SMOVL C00314 BC00314 V=166.7  +MOVJ EC00314
SMOVL C00315 BC00315 V=166.7  +MOVJ EC00315
SREFP 3 C00316 BC00316  +REFP EC00316
CALL JOB:SEARCH-R1-S13D
SET P024 P006
SFTON3D P024
SMOVL C00317 BC00317 V=166.7  +MOVJ EC00317
SMOVL C00318 BC00318 V=166.7  +MOVJ EC00318
SREFP 3 C00319 BC00319  +REFP EC00319
CALL JOB:SEARCH-R1-S13D
SET P024 P006
SFTON3D P024
SMOVL C00320 BC00320 V=166.7  +MOVJ EC00320
MOVL C00321 BC00321 V=1000.0  +MOVJ EC00321 VJ=100.00
MOVL C00322 BC00322 V=1000.0  +MOVJ EC00322 VJ=100.00
'EndPath S3665
'Path S4335
SFTOF3D
MOVJ C00323 BC00323 VJ=100.00  +MOVJ EC00323 VJ=100.00
MOVL C00324 BC00324 V=800.0  +MOVJ EC00324 VJ=100.00
SMOVL C00325 BC00325 V=166.7  +MOVJ EC00325
SREFP 3 C00326 BC00326  +REFP EC00326
CALL JOB:SEARCH-R1-S13D
SET P025 P006
SFTON3D P025
SMOVL C00327 BC00327 V=166.7  +MOVJ EC00327
SMOVL C00328 BC00328 V=166.7  +MOVJ EC00328
SREFP 3 C00329 BC00329  +REFP EC00329
CALL JOB:SEARCH-R1-S13D
SET P025 P006
SFTON3D P025
SMOVL C00330 BC00330 V=166.7  +MOVJ EC00330
SMOVL C00331 BC00331 V=166.7  +MOVJ EC00331
SREFP 3 C00332 BC00332  +REFP EC00332
CALL JOB:SEARCH-R1-S13D
SET P025 P006
SFTON3D P025
SMOVL C00333 BC00333 V=166.7  +MOVJ EC00333
MOVL C00334 BC00334 V=1000.0  +MOVJ EC00334 VJ=100.00
MOVL C00335 BC00335 V=1000.0  +MOVJ EC00335 VJ=100.00
'EndPath S4335
'Path S3666
SFTOF3D
MOVJ C00336 BC00336 VJ=100.00  +MOVJ EC00336 VJ=100.00
MOVL C00337 BC00337 V=800.0  +MOVJ EC00337 VJ=100.00
SMOVL C00338 BC00338 V=166.7  +MOVJ EC00338
SREFP 3 C00339 BC00339  +REFP EC00339
CALL JOB:SEARCH-R1-S13D
SET P026 P006
SFTON3D P026
SMOVL C00340 BC00340 V=166.7  +MOVJ EC00340
SREFP 3 C00341 BC00341  +REFP EC00341
CALL JOB:SEARCH-R1-S13D
SET P026 P006
SFTON3D P026
SMOVL C00342 BC00342 V=166.7  +MOVJ EC00342
MOVL C00343 BC00343 V=1000.0  +MOVJ EC00343 VJ=100.00
'EndPath S3666
MOVJ C00344 BC00344 VJ=100.00  +MOVJ EC00344 VJ=100.00
MOVJ C00345 BC00345 VJ=100.00  +MOVJ EC00345 VJ=100.00
'Path S3661
SFTOF3D
MOVJ C00346 BC00346 VJ=100.00  +MOVJ EC00346 VJ=100.00
MOVL C00347 BC00347 V=800.0  +MOVJ EC00347 VJ=100.00
SMOVL C00348 BC00348 V=166.7  +MOVJ EC00348
SREFP 3 C00349 BC00349  +REFP EC00349
CALL JOB:SEARCH-R1-S13D
SET P027 P006
SFTON3D P027
SMOVL C00350 BC00350 V=166.7  +MOVJ EC00350
SMOVL C00351 BC00351 V=166.7  +MOVJ EC00351
SREFP 3 C00352 BC00352  +REFP EC00352
CALL JOB:SEARCH-R1-S13D
SET P027 P006
SFTON3D P027
SMOVL C00353 BC00353 V=250.0  +MOVJ EC00353
SMOVL C00354 BC00354 V=166.7  +MOVJ EC00354
SREFP 3 C00355 BC00355  +REFP EC00355
CALL JOB:SEARCH-R1-S13D
SET P027 P006
SFTON3D P027
SMOVL C00356 BC00356 V=166.7  +MOVJ EC00356
MOVL C00357 BC00357 V=1000.0  +MOVJ EC00357 VJ=100.00
MOVL C00358 BC00358 V=1000.0  +MOVJ EC00358 VJ=100.00
'EndPath S3661
'Path S4336
SFTOF3D
MOVJ C00359 BC00359 VJ=100.00  +MOVJ EC00359 VJ=100.00
MOVL C00360 BC00360 V=800.0  +MOVJ EC00360 VJ=100.00
SMOVL C00361 BC00361 V=166.7  +MOVJ EC00361
SREFP 3 C00362 BC00362  +REFP EC00362
CALL JOB:SEARCH-R1-S13D
SET P028 P006
SFTON3D P028
SMOVL C00363 BC00363 V=166.7  +MOVJ EC00363
SREFP 3 C00364 BC00364  +REFP EC00364
CALL JOB:SEARCH-R1-S13D
SET P028 P006
SFTON3D P028
SMOVL C00365 BC00365 V=166.7  +MOVJ EC00365
MOVL C00366 BC00366 V=1000.0  +MOVJ EC00366 VJ=100.00
'EndPath S4336
MOVJ C00367 BC00367 VJ=100.00  +MOVJ EC00367 VJ=100.00
'Path S4879
SFTOF3D
MOVJ C00368 BC00368 VJ=100.00  +MOVJ EC00368 VJ=100.00
MOVL C00369 BC00369 V=800.0  +MOVJ EC00369 VJ=100.00
SMOVL C00370 BC00370 V=166.7  +MOVJ EC00370
SREFP 3 C00371 BC00371  +REFP EC00371
CALL JOB:SEARCH-R1-S13D
SET P060 P006
SFTON3D P060
SMOVL C00372 BC00372 V=166.7  +MOVJ EC00372
SMOVL C00373 BC00373 V=166.7  +MOVJ EC00373
SREFP 3 C00374 BC00374  +REFP EC00374
CALL JOB:SEARCH-R1-S13D
SET P060 P006
SFTON3D P060
SMOVL C00375 BC00375 V=166.7  +MOVJ EC00375
SMOVL C00376 BC00376 V=250.0  +MOVJ EC00376
SMOVL C00377 BC00377 V=166.7  +MOVJ EC00377
SREFP 3 C00378 BC00378  +REFP EC00378
CALL JOB:SEARCH-R1-S13D
SET P060 P006
SFTON3D P060
SMOVL C00379 BC00379 V=166.7  +MOVJ EC00379
MOVL C00380 BC00380 V=1000.0  +MOVJ EC00380 VJ=100.00
'EndPath S4879
MOVJ C00381 BC00381 VJ=100.00  +MOVJ EC00381 VJ=100.00
'Path S3664
SFTOF3D
COMM PAUSE
COMM MOVJ C00382 BC00382 VJ=100.00  +MOVJ EC00382 VJ=100.00
COMM MOVL C00383 BC00383 V=800.0  +MOVJ EC00383 VJ=100.00
COMM SMOVL C00384 BC00384 V=166.7  +MOVJ EC00384
COMM SREFP 3 C00385 BC00385  +REFP EC00385
COMM CALL JOB:SEARCH-R1-S13D
COMM SET P029 P006
COMM SFTON3D P029
COMM SMOVL C00386 BC00386 V=166.7  +MOVJ EC00386
COMM SREFP 3 C00387 BC00387  +REFP EC00387
COMM CALL JOB:SEARCH-R1-S13D
COMM SET P029 P006
COMM SFTON3D P029
COMM SMOVL C00388 BC00388 V=166.7  +MOVJ EC00388
COMM MOVL C00389 BC00389 V=1000.0  +MOVJ EC00389 VJ=100.00
COMM 'EndPath S3664
COMM 'Path S4337
COMM SFTOF3D
COMM MOVJ C00390 BC00390 VJ=100.00  +MOVJ EC00390 VJ=100.00
COMM MOVL C00391 BC00391 V=800.0  +MOVJ EC00391 VJ=100.00
COMM SMOVL C00392 BC00392 V=166.7  +MOVJ EC00392
COMM SREFP 3 C00393 BC00393  +REFP EC00393
COMM CALL JOB:SEARCH-R1-S13D
COMM SET P030 P006
COMM SFTON3D P030
COMM SMOVL C00394 BC00394 V=166.7  +MOVJ EC00394
COMM SREFP 3 C00395 BC00395  +REFP EC00395
COMM CALL JOB:SEARCH-R1-S13D
COMM SET P030 P006
COMM SFTON3D P030
COMM SMOVL C00396 BC00396 V=166.7  +MOVJ EC00396
COMM MOVL C00397 BC00397 V=800.0  +MOVJ EC00397 VJ=100.00
COMM MOVL C00398 BC00398 V=1000.0  +MOVJ EC00398 VJ=100.00
COMM 'EndPath S4337
MOVJ C00399 BC00399 VJ=100.00  +MOVJ EC00399 VJ=100.00
'Path S3663
SFTOF3D
MOVJ C00400 BC00400 VJ=100.00  +MOVJ EC00400 VJ=100.00
MOVL C00401 BC00401 V=800.0  +MOVJ EC00401 VJ=100.00
SMOVL C00402 BC00402 V=166.7  +MOVJ EC00402
SREFP 3 C00403 BC00403  +REFP EC00403
CALL JOB:SEARCH-R1-S13D
SET P031 P006
SFTON3D P031
SMOVL C00404 BC00404 V=166.7  +MOVJ EC00404
SREFP 3 C00405 BC00405  +REFP EC00405
CALL JOB:SEARCH-R1-S13D
SET P031 P006
SFTON3D P031
SMOVL C00406 BC00406 V=166.7  +MOVJ EC00406
SMOVL C00407 BC00407 V=166.7  +MOVJ EC00407
SREFP 3 C00408 BC00408  +REFP EC00408
CALL JOB:SEARCH-R1-S13D
SET P031 P006
SFTON3D P031
SMOVL C00409 BC00409 V=166.7  +MOVJ EC00409
MOVL C00410 BC00410 V=1000.0  +MOVJ EC00410 VJ=100.00
'EndPath S3663
MOVJ C00411 BC00411 VJ=100.00  +MOVJ EC00411 VJ=100.00
'Path S4338
SFTOF3D
MOVJ C00412 BC00412 VJ=100.00  +MOVJ EC00412 VJ=100.00
MOVL C00413 BC00413 V=800.0  +MOVJ EC00413 VJ=100.00
SMOVL C00414 BC00414 V=166.7  +MOVJ EC00414
SREFP 3 C00415 BC00415  +REFP EC00415
CALL JOB:SEARCH-R1-S13D
SET P032 P006
SFTON3D P032
SMOVL C00416 BC00416 V=166.7  +MOVJ EC00416
SREFP 3 C00417 BC00417  +REFP EC00417
CALL JOB:SEARCH-R1-S13D
SET P032 P006
SFTON3D P032
SMOVL C00418 BC00418 V=166.7  +MOVJ EC00418
SMOVL C00419 BC00419 V=166.7  +MOVJ EC00419
SREFP 3 C00420 BC00420  +REFP EC00420
CALL JOB:SEARCH-R1-S13D
SET P032 P006
SFTON3D P032
SMOVL C00421 BC00421 V=166.7  +MOVJ EC00421
MOVL C00422 BC00422 V=1000.0  +MOVJ EC00422 VJ=100.00
'EndPath S4338
MOVJ C00423 BC00423 VJ=100.00  +MOVJ EC00423 VJ=100.00
'Path S3662
SFTOF3D
MOVJ C00424 BC00424 VJ=100.00  +MOVJ EC00424 VJ=100.00
MOVL C00425 BC00425 V=800.0  +MOVJ EC00425 VJ=100.00
SMOVL C00426 BC00426 V=166.7  +MOVJ EC00426
SREFP 3 C00427 BC00427  +REFP EC00427
CALL JOB:SEARCH-R1-S13D
SET P033 P006
SFTON3D P033
SMOVL C00428 BC00428 V=166.7  +MOVJ EC00428
SREFP 3 C00429 BC00429  +REFP EC00429
CALL JOB:SEARCH-R1-S13D
SET P033 P006
SFTON3D P033
SMOVL C00430 BC00430 V=166.7  +MOVJ EC00430
MOVL C00431 BC00431 V=1000.0  +MOVJ EC00431 VJ=100.00
'EndPath S3662
'Path S4339
SFTOF3D
MOVJ C00432 BC00432 VJ=100.00  +MOVJ EC00432 VJ=100.00
MOVL C00433 BC00433 V=800.0  +MOVJ EC00433 VJ=100.00
SMOVL C00434 BC00434 V=166.7  +MOVJ EC00434
SREFP 3 C00435 BC00435  +REFP EC00435
CALL JOB:SEARCH-R1-S13D
SET P034 P006
SFTON3D P034
SMOVL C00436 BC00436 V=166.7  +MOVJ EC00436
SMOVL C00437 BC00437 V=166.7  +MOVJ EC00437
SREFP 3 C00438 BC00438  +REFP EC00438
CALL JOB:SEARCH-R1-S13D
SET P034 P006
SFTON3D P034
SMOVL C00439 BC00439 V=166.7  +MOVJ EC00439
SMOVL C00440 BC00440 V=166.7  +MOVJ EC00440
SREFP 3 C00441 BC00441  +REFP EC00441
CALL JOB:SEARCH-R1-S13D
SET P034 P006
SFTON3D P034
SMOVL C00442 BC00442 V=166.7  +MOVJ EC00442
MOVL C00443 BC00443 V=1000.0  +MOVJ EC00443 VJ=100.00
'EndPath S4339
MOVJ C00444 BC00444 VJ=100.00  +MOVJ EC00444 VJ=100.00
'Path W3667
SFTOF3D
SFTON3D P026
MOVJ C00445 BC00445 VJ=100.00  +MOVJ EC00445 VJ=100.00
SMOVL C00446 BC00446 V=800.0  +MOVJ EC00446
SREFP 1 C00447 BC00447  +REFP EC00447
SREFP 2 C00448 BC00448  +REFP EC00448
SMOVL C00449 BC00449 V=166.7 PL=0  +MOVJ EC00449
MACRO1 MJ#(0) ARGF21
ARCON
SWVON WEV#(100)
SMOVL C00450 BC00450 V=9.2  +MOVJ EC00450
SMOVL C00451 BC00451 V=9.2  +MOVJ EC00451
SMOVL C00452 BC00452 V=9.2  +MOVJ EC00452
ARCOF
SWVOF
SMOVL C00453 BC00453 V=800.0  +MOVJ EC00453
SMOVL C00454 BC00454 V=1000.0  +MOVJ EC00454
SFTOF3D
'EndPath W3667
MOVJ C00455 BC00455 VJ=100.00  +MOVJ EC00455 VJ=100.00
MOVJ C00456 BC00456 VJ=100.00  +MOVJ EC00456 VJ=100.00
'Path W3668
SSFTOF
SFTOF3D
SFTON3D P028
MOVJ C00457 BC00457 VJ=100.00  +MOVJ EC00457 VJ=100.00
SMOVL C00458 BC00458 V=800.0  +MOVJ EC00458
SREFP 1 C00459 BC00459  +REFP EC00459
SREFP 2 C00460 BC00460  +REFP EC00460
SMOVL C00461 BC00461 V=150.0 PL=0  +MOVJ EC00461
ARCON
SWVON WEV#(100)
SFTON3D P027
SMOVL C00462 BC00462 V=9.2  +MOVJ EC00462
SMOVL C00463 BC00463 V=9.2  +MOVJ EC00463
ARCOF
SWVOF
SMOVL C00464 BC00464 V=800.0  +MOVJ EC00464
SMOVL C00465 BC00465 V=1000.0  +MOVJ EC00465
SFTOF3D
'EndPath W3668
MOVJ C00466 BC00466 VJ=100.00  +MOVJ EC00466 VJ=100.00
COMM 'Path W4546
COMM PAUSE
COMM SFTOF3D
COMM SFTON3D P022
COMM MOVJ C00467 BC00467 VJ=100.00  +MOVJ EC00467 VJ=100.00
COMM SMOVL C00468 BC00468 V=800.0  +MOVJ EC00468
COMM SMOVL C00469 BC00469 V=150.0 PL=0  +MOVJ EC00469
COMM MACRO1 MJ#(0) ARGF9
COMM ARCON
COMM SWVON WEV#(10)
COMM SFTON3D P021
COMM SMOVL C00470 BC00470 V=10.0  +MOVJ EC00470
COMM ARCOF
COMM SWVOF
COMM SMOVL C00471 BC00471 V=800.0  +MOVJ EC00471
COMM SMOVL C00472 BC00472 V=1000.0  +MOVJ EC00472
COMM SFTOF3D
COMM 'EndPath W4546
COMM 'Path W4901
COMM SFTOF3D
SFTON3D P060
COMM MOVJ C00473 BC00473 VJ=100.00  +MOVJ EC00473 VJ=100.00
MOVJ C00474 BC00474 VJ=100.00  +MOVJ EC00474 VJ=100.00
MOVJ C00475 BC00475 VJ=100.00  +MOVJ EC00475 VJ=100.00
SMOVL C00476 BC00476 V=800.0  +MOVJ EC00476
SMOVL C00477 BC00477 V=150.0 PL=0  +MOVJ EC00477
MACRO1 MJ#(0) ARGF14
ARCON
SMOVL C00478 BC00478 V=10.8  +MOVJ EC00478
ARCOF
SMOVL C00479 BC00479 V=800.0  +MOVJ EC00479
SFTOF3D
'EndPath W4901
'Path W4880
SFTOF3D
SFTON3D P060
SMOVL C00480 BC00480 V=800.0  +MOVJ EC00480
SMOVL C00481 BC00481 V=150.0 PL=0  +MOVJ EC00481
ARCON
SMOVL C00482 BC00482 V=10.0  +MOVJ EC00482
SMOVL C00483 BC00483 V=10.0  +MOVJ EC00483
SMOVL C00484 BC00484 V=10.0  +MOVJ EC00484
ARCOF
SMOVL C00485 BC00485 V=800.0  +MOVJ EC00485
SMOVL C00486 BC00486 V=1000.0  +MOVJ EC00486
SFTOF3D
'EndPath W4880
MOVJ C00487 BC00487 VJ=100.00  +MOVJ EC00487 VJ=100.00
COMM PAUSE
COMM MOVJ C00488 BC00488 VJ=100.00  +MOVJ EC00488 VJ=100.00
COMM 'Path W4548
COMM SFTOF3D
COMM SFTON3D P030
COMM MOVJ C00489 BC00489 VJ=100.00  +MOVJ EC00489 VJ=100.00
COMM SMOVL C00490 BC00490 V=800.0  +MOVJ EC00490
COMM SMOVL C00491 BC00491 V=150.0 PL=0  +MOVJ EC00491
COMM MACRO1 MJ#(0) ARGF9
COMM ARCON
COMM SFTON3D P029
COMM SMOVL C00492 BC00492 V=10.0  +MOVJ EC00492
COMM SMOVL C00493 BC00493 V=10.0  +MOVJ EC00493
COMM ARCOF
COMM SMOVL C00494 BC00494 V=800.0  +MOVJ EC00494
COMM SMOVL C00495 BC00495 V=1000.0  +MOVJ EC00495
COMM SFTOF3D
COMM 'EndPath W4548
COMM MOVJ C00496 BC00496 VJ=100.00  +MOVJ EC00496 VJ=100.00
MOVJ C00497 BC00497 VJ=100.00  +MOVJ EC00497 VJ=100.00
'Path W3671
SFTOF3D
SFTON3D P033
MOVJ C00498 BC00498 VJ=100.00  +MOVJ EC00498 VJ=100.00
SMOVL C00499 BC00499 V=800.0  +MOVJ EC00499
SMOVL C00500 BC00500 V=166.7 PL=0  +MOVJ EC00500
MACRO1 MJ#(0) ARGF14
ARCON
SMOVL C00501 BC00501 V=9.2  +MOVJ EC00501
SFTON3D P034
SMOVL C00502 BC00502 V=9.2  +MOVJ EC00502
SMOVL C00503 BC00503 V=9.2  +MOVJ EC00503
ARCOF
SMOVL C00504 BC00504 V=800.0  +MOVJ EC00504
SMOVL C00505 BC00505 V=1000.0  +MOVJ EC00505
SFTOF3D
'EndPath W3671
MOVJ C00506 BC00506 VJ=100.00  +MOVJ EC00506 VJ=100.00
'Path W3672
SFTOF3D
SFTON3D P024
MOVJ C00507 BC00507 VJ=100.00  +MOVJ EC00507 VJ=100.00
SMOVL C00508 BC00508 V=800.0  +MOVJ EC00508
SMOVL C00509 BC00509 V=166.7 PL=0  +MOVJ EC00509
ARCON
SMOVL C00510 BC00510 V=9.2  +MOVJ EC00510
SFTON3D P025
SMOVL C00511 BC00511 V=9.2  +MOVJ EC00511
SMOVL C00512 BC00512 V=9.2  +MOVJ EC00512
ARCOF
SMOVL C00513 BC00513 V=800.0  +MOVJ EC00513
SMOVL C00514 BC00514 V=1000.0  +MOVJ EC00514
SFTOF3D
'EndPath W3672
MOVJ C00515 BC00515 VJ=100.00  +MOVJ EC00515 VJ=100.00
'Path W3673
SFTOF3D
SFTON3D P032
MOVJ C00516 BC00516 VJ=100.00  +MOVJ EC00516 VJ=100.00
SMOVL C00517 BC00517 V=800.0  +MOVJ EC00517
SMOVL C00518 BC00518 V=166.7 PL=0  +MOVJ EC00518
ARCON
SMOVL C00519 BC00519 V=9.2  +MOVJ EC00519
SFTON3D P031
SMOVL C00520 BC00520 V=9.2  +MOVJ EC00520
SMOVL C00521 BC00521 V=9.2  +MOVJ EC00521
ARCOF
SMOVL C00522 BC00522 V=800.0  +MOVJ EC00522
SMOVL C00523 BC00523 V=1000.0  +MOVJ EC00523
SFTOF3D
'EndPath W3673
MOVJ C00524 BC00524 VJ=100.00  +MOVJ EC00524 VJ=100.00
'
MOVJ C00525 BC00525 VJ=100.00  +MOVJ EC00525 VJ=100.00
JUMP *VV
MOVJ C00526 BC00526 VJ=100.00  +MOVJ EC00526 VJ=100.00
'Path W3680
SFTOF3D
SFTON3D P023
MOVJ C00527 BC00527 VJ=100.00  +MOVJ EC00527 VJ=100.00
SMOVL C00528 BC00528 V=800.0  +MOVJ EC00528
SMOVL C00529 BC00529 V=166.7 PL=0  +MOVJ EC00529
SMOVL C00530 BC00530 V=10.0  +MOVJ EC00530
SMOVL C00531 BC00531 V=33.3  +MOVJ EC00531
SMOVL C00532 BC00532 V=33.3  +MOVJ EC00532
SMOVL C00533 BC00533 V=33.3  +MOVJ EC00533
SMOVL C00534 BC00534 V=10.0  +MOVJ EC00534
SMOVL C00535 BC00535 V=10.0  +MOVJ EC00535
SMOVL C00536 BC00536 V=10.0  +MOVJ EC00536
SMOVL C00537 BC00537 V=10.0  +MOVJ EC00537
SMOVL C00538 BC00538 V=10.0  +MOVJ EC00538
ARCOF
SMOVL C00539 BC00539 V=800.0  +MOVJ EC00539
SMOVL C00540 BC00540 V=1000.0  +MOVJ EC00540
SFTOF3D
'EndPath W3680
'Path W3681
*VV
SFTOF3D
SFTON3D P023
MOVJ C00541 BC00541 VJ=100.00  +MOVJ EC00541 VJ=100.00
SMOVL C00542 BC00542 V=800.0  +MOVJ EC00542
MACRO1 MJ#(0) ARGF9
SMOVL C00543 BC00543 V=166.7 PL=0  +MOVJ EC00543
COMM SMOVL C00544 BC00544 V=150.0 PL=0  +MOVJ EC00544
COMM MACRO1 MJ#(0) ARGF9
COMM ARCON
COMM SMOVL C00545 BC00545 V=8.3  +MOVJ EC00545
COMM SMOVL C00546 BC00546 V=8.3  +MOVJ EC00546
COMM SMOVL C00547 BC00547 V=8.3  +MOVJ EC00547
ARCON
SMOVL C00548 BC00548 V=8.3  +MOVJ EC00548
SMOVL C00549 BC00549 V=8.3  +MOVJ EC00549
SMOVL C00550 BC00550 V=8.3  +MOVJ EC00550
SMOVL C00551 BC00551 V=8.3  +MOVJ EC00551
SMOVL C00552 BC00552 V=8.3  +MOVJ EC00552
SMOVL C00553 BC00553 V=8.3  +MOVJ EC00553
ARCOF
SMOVL C00554 BC00554 V=800.0  +MOVJ EC00554
SMOVL C00555 BC00555 V=1000.0  +MOVJ EC00555
SFTOF3D
'EndPath W3681
'Down
MOVJ C00556 BC00556 VJ=100.00  +MOVJ EC00556 VJ=100.00
CALL JOB:CLEAN-R1_KM_3P
'1
MOVJ C00557 BC00557 VJ=100.00  +MOVJ EC00557 VJ=100.00
MOVJ C00558 BC00558 VJ=100.00  +MOVJ EC00558 VJ=100.00
MOVJ C00559 BC00559 VJ=100.00  +MOVJ EC00559 VJ=100.00
'Path S4334
SFTOF3D
MOVJ C00560 BC00560 VJ=100.00  +MOVJ EC00560 VJ=100.00
MOVL C00561 BC00561 V=800.0  +MOVJ EC00561 VJ=100.00
SMOVL C00562 BC00562 V=166.7  +MOVJ EC00562
SREFP 3 C00563 BC00563  +REFP EC00563
CALL JOB:SEARCH-R1-S13D
SET P048 P006
SFTON3D P048
SMOVL C00564 BC00564 V=166.7  +MOVJ EC00564
SMOVL C00565 BC00565 V=166.7  +MOVJ EC00565
SREFP 3 C00566 BC00566  +REFP EC00566
CALL JOB:SEARCH-R1-S13D
SET P048 P006
SFTON3D P048
SMOVL C00567 BC00567 V=166.7  +MOVJ EC00567
MOVL C00568 BC00568 V=1000.0  +MOVJ EC00568 VJ=100.00
'EndPath S4334
'Path S4335
SFTOF3D
MOVJ C00569 BC00569 VJ=100.00  +MOVJ EC00569 VJ=100.00
MOVL C00570 BC00570 V=800.0  +MOVJ EC00570 VJ=100.00
SMOVL C00571 BC00571 V=166.7  +MOVJ EC00571
SREFP 3 C00572 BC00572  +REFP EC00572
CALL JOB:SEARCH-R1-S13D
SET P047 P006
SFTON3D P047
SMOVL C00573 BC00573 V=250.0  +MOVJ EC00573
SMOVL C00574 BC00574 V=166.7  +MOVJ EC00574
SREFP 3 C00575 BC00575  +REFP EC00575
CALL JOB:SEARCH-R1-S13D
SET P047 P006
SFTON3D P047
SMOVL C00576 BC00576 V=166.7  +MOVJ EC00576
MOVL C00577 BC00577 V=1000.0  +MOVJ EC00577 VJ=100.00
'EndPath S4335
MOVJ C00578 BC00578 VJ=100.00  +MOVJ EC00578 VJ=100.00
MOVJ C00579 BC00579 VJ=100.00  +MOVJ EC00579 VJ=100.00
MOVJ C00580 BC00580 VJ=100.00  +MOVJ EC00580 VJ=100.00
MOVJ C00581 BC00581 VJ=100.00  +MOVJ EC00581 VJ=100.00
'Path S4336
SFTOF3D
MOVJ C00582 BC00582 VJ=100.00  +MOVJ EC00582 VJ=100.00
MOVL C00583 BC00583 V=800.0  +MOVJ EC00583 VJ=100.00
SMOVL C00584 BC00584 V=166.7  +MOVJ EC00584
SREFP 3 C00585 BC00585  +REFP EC00585
CALL JOB:SEARCH-R1-S13D
SET P046 P006
SFTON3D P046
SMOVL C00586 BC00586 V=250.0  +MOVJ EC00586
SMOVL C00587 BC00587 V=166.7  +MOVJ EC00587
SREFP 3 C00588 BC00588  +REFP EC00588
CALL JOB:SEARCH-R1-S13D
SET P046 P006
SFTON3D P046
SMOVL C00589 BC00589 V=166.7  +MOVJ EC00589
MOVL C00590 BC00590 V=1000.0  +MOVJ EC00590 VJ=100.00
'EndPath S4336
'Path S4337
SFTOF3D
MOVJ C00591 BC00591 VJ=100.00  +MOVJ EC00591 VJ=100.00
MOVL C00592 BC00592 V=800.0  +MOVJ EC00592 VJ=100.00
SMOVL C00593 BC00593 V=166.7  +MOVJ EC00593
SREFP 3 C00594 BC00594  +REFP EC00594
CALL JOB:SEARCH-R1-S13D
SET P050 P006
SFTON3D P050
SMOVL C00595 BC00595 V=166.7  +MOVJ EC00595
SREFP 3 C00596 BC00596  +REFP EC00596
CALL JOB:SEARCH-R1-S13D
SET P050 P006
SFTON3D P050
SMOVL C00597 BC00597 V=166.7  +MOVJ EC00597
MOVL C00598 BC00598 V=1000.0  +MOVJ EC00598 VJ=100.00
'EndPath S4337
'Path S4338
SFTOF3D
MOVJ C00599 BC00599 VJ=100.00  +MOVJ EC00599 VJ=100.00
MOVL C00600 BC00600 V=666.7  +MOVJ EC00600 VJ=100.00
SMOVL C00601 BC00601 V=166.7  +MOVJ EC00601
SREFP 3 C00602 BC00602  +REFP EC00602
CALL JOB:SEARCH-R1-S13D
SET P051 P006
SFTON3D P051
SMOVL C00603 BC00603 V=166.7  +MOVJ EC00603
SREFP 3 C00604 BC00604  +REFP EC00604
CALL JOB:SEARCH-R1-S13D
SET P051 P006
SFTON3D P051
SMOVL C00605 BC00605 V=166.7  +MOVJ EC00605
SMOVL C00606 BC00606 V=166.7  +MOVJ EC00606
SMOVL C00607 BC00607 V=133.3  +MOVJ EC00607
SREFP 3 C00608 BC00608  +REFP EC00608
CALL JOB:SEARCH-R1-S13D
SET P051 P006
SFTON3D P051
SMOVL C00609 BC00609 V=250.0  +MOVJ EC00609
SMOVL C00610 BC00610 V=500.0  +MOVJ EC00610
'EndPath S4338
'Path S4339
SFTOF3D
MOVJ C00611 BC00611 VJ=100.00  +MOVJ EC00611 VJ=100.00
MOVL C00612 BC00612 V=800.0  +MOVJ EC00612 VJ=100.00
SMOVL C00613 BC00613 V=166.7  +MOVJ EC00613
SREFP 3 C00614 BC00614  +REFP EC00614
CALL JOB:SEARCH-R1-S13D
SET P045 P006
SFTON3D P045
SMOVL C00615 BC00615 V=250.0  +MOVJ EC00615
SMOVL C00616 BC00616 V=166.7  +MOVJ EC00616
SREFP 3 C00617 BC00617  +REFP EC00617
CALL JOB:SEARCH-R1-S13D
SET P045 P006
SFTON3D P045
SMOVL C00618 BC00618 V=166.7  +MOVJ EC00618
MOVL C00619 BC00619 V=1000.0  +MOVJ EC00619 VJ=100.00
'EndPath S4339
'Path S4340
SFTOF3D
MOVJ C00620 BC00620 VJ=100.00  +MOVJ EC00620 VJ=100.00
MOVL C00621 BC00621 V=800.0  +MOVJ EC00621 VJ=100.00
SMOVL C00622 BC00622 V=166.7  +MOVJ EC00622
SREFP 3 C00623 BC00623  +REFP EC00623
CALL JOB:SEARCH-R1-S13D
SET P044 P006
SFTON3D P044
SMOVL C00624 BC00624 V=250.0  +MOVJ EC00624
SMOVL C00625 BC00625 V=166.7  +MOVJ EC00625
SREFP 3 C00626 BC00626  +REFP EC00626
CALL JOB:SEARCH-R1-S13D
SET P044 P006
SFTON3D P044
SMOVL C00627 BC00627 V=166.7  +MOVJ EC00627
MOVL C00628 BC00628 V=1000.0  +MOVJ EC00628 VJ=100.00
'EndPath S4340
'Path S4341
SFTOF3D
MOVJ C00629 BC00629 VJ=100.00  +MOVJ EC00629 VJ=100.00
MOVL C00630 BC00630 V=800.0  +MOVJ EC00630 VJ=100.00
SMOVL C00631 BC00631 V=166.7  +MOVJ EC00631
SREFP 3 C00632 BC00632  +REFP EC00632
CALL JOB:SEARCH-R1-S13D
SET P049 P006
SFTON3D P049
SMOVL C00633 BC00633 V=166.7  +MOVJ EC00633
SMOVL C00634 BC00634 V=166.7  +MOVJ EC00634
SREFP 3 C00635 BC00635  +REFP EC00635
CALL JOB:SEARCH-R1-S13D
SET P049 P006
SFTON3D P049
SMOVL C00636 BC00636 V=166.7  +MOVJ EC00636
MOVL C00637 BC00637 V=1000.0  +MOVJ EC00637 VJ=100.00
'EndPath S4341
MOVJ C00638 BC00638 VJ=100.00  +MOVJ EC00638 VJ=100.00
MOVJ C00639 BC00639 VJ=100.00  +MOVJ EC00639 VJ=100.00
'Path S4342
SFTOF3D
MOVJ C00640 BC00640 VJ=100.00  +MOVJ EC00640 VJ=100.00
MOVL C00641 BC00641 V=800.0  +MOVJ EC00641 VJ=100.00
SMOVL C00642 BC00642 V=166.7  +MOVJ EC00642
SREFP 3 C00643 BC00643  +REFP EC00643
CALL JOB:SEARCH-R1-S13D
SET P043 P006
SFTON3D P043
SMOVL C00644 BC00644 V=166.7  +MOVJ EC00644
SMOVL C00645 BC00645 V=166.7  +MOVJ EC00645
SREFP 3 C00646 BC00646  +REFP EC00646
CALL JOB:SEARCH-R1-S13D
SET P043 P006
SFTON3D P043
SMOVL C00647 BC00647 V=166.7  +MOVJ EC00647
MOVL C00648 BC00648 V=1000.0  +MOVJ EC00648 VJ=100.00
'EndPath S4342
'Path S4343
SFTOF3D
MOVJ C00649 BC00649 VJ=100.00  +MOVJ EC00649 VJ=100.00
MOVL C00650 BC00650 V=800.0  +MOVJ EC00650 VJ=100.00
SMOVL C00651 BC00651 V=166.7  +MOVJ EC00651
SREFP 3 C00652 BC00652  +REFP EC00652
CALL JOB:SEARCH-R1-S13D
SET P042 P006
SFTON3D P042
SMOVL C00653 BC00653 V=250.0  +MOVJ EC00653
SMOVL C00654 BC00654 V=166.7  +MOVJ EC00654
SREFP 3 C00655 BC00655  +REFP EC00655
CALL JOB:SEARCH-R1-S13D
SET P042 P006
SFTON3D P042
SMOVL C00656 BC00656 V=166.7  +MOVJ EC00656
MOVL C00657 BC00657 V=1000.0  +MOVJ EC00657 VJ=100.00
'EndPath S4343
MOVJ C00658 BC00658 VJ=100.00  +MOVJ EC00658 VJ=100.00
'
'Path W4344
SFTOF3D
SFTON3D P051
MOVJ C00659 BC00659 VJ=60.00  +MOVJ EC00659 VJ=20.00
SMOVL C00660 BC00660 V=500.0  +MOVJ EC00660
SMOVL C00661 BC00661 V=166.7 PL=0  +MOVJ EC00661
MACRO1 MJ#(0) ARGF14
ARCON
SMOVL C00662 BC00662 V=8.3  +MOVJ EC00662
ARCOF
SMOVL C00663 BC00663 V=800.0  +MOVJ EC00663
SMOVL C00664 BC00664 V=150.0  +MOVJ EC00664
ARCON
SMOVL C00665 BC00665 V=11.7  +MOVJ EC00665
ARCOF
SMOVL C00666 BC00666 V=250.0  +MOVJ EC00666
SMOVL C00667 BC00667 V=500.0  +MOVJ EC00667
SMOVL C00668 BC00668 V=1000.0  +MOVJ EC00668
SFTOF3D
'EndPath W4344
'Path W4345
SFTOF3D
SFTON3D P045
MOVJ C00669 BC00669 VJ=100.00  +MOVJ EC00669 VJ=100.00
SMOVL C00670 BC00670 V=800.0  +MOVJ EC00670
SMOVL C00671 BC00671 V=150.0 PL=0  +MOVJ EC00671
MACRO1 MJ#(0) ARGF21
ARCON
SMOVL C00672 BC00672 V=11.7  +MOVJ EC00672
ARCOF
SMOVL C00673 BC00673 V=800.0  +MOVJ EC00673
SMOVL C00674 BC00674 V=1000.0  +MOVJ EC00674
SFTOF3D
'EndPath W4345
'Path W4346
SFTOF3D
SFTON3D P045
MOVJ C00675 BC00675 VJ=100.00  +MOVJ EC00675 VJ=100.00
SMOVL C00676 BC00676 V=800.0  +MOVJ EC00676
SMOVL C00677 BC00677 V=150.0 PL=0  +MOVJ EC00677
ARCON
SMOVL C00678 BC00678 V=11.7  +MOVJ EC00678
ARCOF
SMOVL C00679 BC00679 V=800.0  +MOVJ EC00679
SMOVL C00680 BC00680 V=1000.0  +MOVJ EC00680
SFTOF3D
'EndPath W4346
'Path W4347
SFTOF3D
SFTON3D P049
MOVJ C00681 BC00681 VJ=100.00  +MOVJ EC00681 VJ=100.00
SMOVL C00682 BC00682 V=800.0  +MOVJ EC00682
SMOVL C00683 BC00683 V=150.0 PL=0  +MOVJ EC00683
ARCON
SMOVL C00684 BC00684 V=11.7  +MOVJ EC00684
ARCOF
SMOVL C00685 BC00685 V=800.0  +MOVJ EC00685
SMOVL C00686 BC00686 V=1000.0  +MOVJ EC00686
SFTOF3D
'EndPath W4347
'Path W4348
SFTOF3D
SFTON3D P050
MOVJ C00687 BC00687 VJ=100.00  +MOVJ EC00687 VJ=100.00
SMOVL C00688 BC00688 V=800.0  +MOVJ EC00688
SMOVL C00689 BC00689 V=150.0 PL=0  +MOVJ EC00689
ARCON
SMOVL C00690 BC00690 V=11.7  +MOVJ EC00690
ARCOF
SMOVL C00691 BC00691 V=800.0  +MOVJ EC00691
SMOVL C00692 BC00692 V=1000.0  +MOVJ EC00692
SFTOF3D
'EndPath W4348
MOVJ C00693 BC00693 VJ=100.00  +MOVJ EC00693 VJ=100.00
MOVJ C00694 BC00694 VJ=100.00  +MOVJ EC00694 VJ=100.00
'1
'uwaga na podajnik
'Path W4349
SFTOF3D
SFTON3D P048
MOVJ C00695 BC00695 VJ=100.00  +MOVJ EC00695 VJ=100.00
SMOVL C00696 BC00696 V=800.0  +MOVJ EC00696
SMOVL C00697 BC00697 V=150.0 PL=0  +MOVJ EC00697
ARCON
SMOVL C00698 BC00698 V=11.7  +MOVJ EC00698
ARCOF
SMOVL C00699 BC00699 V=800.0  +MOVJ EC00699
SMOVL C00700 BC00700 V=1000.0  +MOVJ EC00700
SFTOF3D
'EndPath W4349
'Path W4350
SFTOF3D
SFTON3D P048
MOVJ C00701 BC00701 VJ=100.00  +MOVJ EC00701 VJ=100.00
SMOVL C00702 BC00702 V=800.0  +MOVJ EC00702
SMOVL C00703 BC00703 V=150.0 PL=0  +MOVJ EC00703
ARCON
SMOVL C00704 BC00704 V=11.7  +MOVJ EC00704
ARCOF
SMOVL C00705 BC00705 V=800.0  +MOVJ EC00705
SMOVL C00706 BC00706 V=1000.0  +MOVJ EC00706
SFTOF3D
'EndPath W4350
'Path W4351
SFTOF3D
SFTON3D P047
MOVJ C00707 BC00707 VJ=100.00  +MOVJ EC00707 VJ=100.00
SMOVL C00708 BC00708 V=800.0  +MOVJ EC00708
SMOVL C00709 BC00709 V=150.0 PL=0  +MOVJ EC00709
ARCON
SMOVL C00710 BC00710 V=11.7  +MOVJ EC00710
ARCOF
SMOVL C00711 BC00711 V=800.0  +MOVJ EC00711
SMOVL C00712 BC00712 V=1000.0  +MOVJ EC00712
SFTOF3D
'EndPath W4351
'2
MOVJ C00713 BC00713 VJ=100.00  +MOVJ EC00713 VJ=100.00
MOVJ C00714 BC00714 VJ=100.00  +MOVJ EC00714 VJ=100.00
'Path W4352
SFTOF3D
SFTON3D P043
MOVJ C00715 BC00715 VJ=100.00  +MOVJ EC00715 VJ=100.00
SMOVL C00716 BC00716 V=800.0  +MOVJ EC00716
SMOVL C00717 BC00717 V=150.0 PL=0  +MOVJ EC00717
ARCON
SMOVL C00718 BC00718 V=11.7  +MOVJ EC00718
ARCOF
SMOVL C00719 BC00719 V=800.0  +MOVJ EC00719
SMOVL C00720 BC00720 V=1000.0  +MOVJ EC00720
SFTOF3D
'EndPath W4352
'Path W4353
SFTOF3D
SFTON3D P043
MOVJ C00721 BC00721 VJ=100.00  +MOVJ EC00721 VJ=100.00
SMOVL C00722 BC00722 V=800.0  +MOVJ EC00722
SMOVL C00723 BC00723 V=150.0 PL=0  +MOVJ EC00723
ARCON
SMOVL C00724 BC00724 V=11.7  +MOVJ EC00724
ARCOF
SMOVL C00725 BC00725 V=800.0  +MOVJ EC00725
SMOVL C00726 BC00726 V=1000.0  +MOVJ EC00726
SFTOF3D
'EndPath W4353
'Path W4354
SFTOF3D
SFTON3D P042
MOVJ C00727 BC00727 VJ=100.00  +MOVJ EC00727 VJ=100.00
SMOVL C00728 BC00728 V=800.0  +MOVJ EC00728
SMOVL C00729 BC00729 V=150.0 PL=0  +MOVJ EC00729
ARCON
SMOVL C00730 BC00730 V=11.7  +MOVJ EC00730
ARCOF
SMOVL C00731 BC00731 V=800.0  +MOVJ EC00731
SMOVL C00732 BC00732 V=1000.0  +MOVJ EC00732
SFTOF3D
'EndPath W4354
'Path W4355
SFTOF3D
SFTON3D P042
MOVJ C00733 BC00733 VJ=100.00  +MOVJ EC00733 VJ=100.00
SMOVL C00734 BC00734 V=800.0  +MOVJ EC00734
SMOVL C00735 BC00735 V=150.0 PL=0  +MOVJ EC00735
ARCON
SMOVL C00736 BC00736 V=11.7  +MOVJ EC00736
ARCOF
SMOVL C00737 BC00737 V=800.0  +MOVJ EC00737
SMOVL C00738 BC00738 V=1000.0  +MOVJ EC00738
SFTOF3D
'EndPath W4355
'3
MOVJ C00739 BC00739 VJ=100.00  +MOVJ EC00739 VJ=100.00
'Path W4356
SFTOF3D
SFTON3D P044
MOVJ C00740 BC00740 VJ=100.00  +MOVJ EC00740 VJ=100.00
SMOVL C00741 BC00741 V=800.0  +MOVJ EC00741
SMOVL C00742 BC00742 V=150.0 PL=0  +MOVJ EC00742
ARCON
SMOVL C00743 BC00743 V=11.7  +MOVJ EC00743
ARCOF
SMOVL C00744 BC00744 V=800.0  +MOVJ EC00744
SMOVL C00745 BC00745 V=1000.0  +MOVJ EC00745
SFTOF3D
'EndPath W4356
'Path W4357
SFTOF3D
SFTON3D P046
MOVJ C00746 BC00746 VJ=100.00  +MOVJ EC00746 VJ=100.00
SMOVL C00747 BC00747 V=800.0  +MOVJ EC00747
SMOVL C00748 BC00748 V=150.0 PL=0  +MOVJ EC00748
MACRO1 MJ#(0) ARGF14
ARCON
SMOVL C00749 BC00749 V=11.7  +MOVJ EC00749
ARCOF
SMOVL C00750 BC00750 V=800.0  +MOVJ EC00750
SMOVL C00751 BC00751 V=1000.0  +MOVJ EC00751
SFTOF3D
'EndPath W4357
MOVJ C00752 BC00752 VJ=100.00  +MOVJ EC00752 VJ=100.00
MOVJ C00753 BC00753 VJ=100.00  +MOVJ EC00753 VJ=100.00
MOVJ C00754 BC00754 VJ=100.00  +MOVJ EC00754 VJ=100.00
END
